Fanuc KAREL source: kb00041.KL

-- PROVISIONAL review KL for V1013-1; original PC SHA256 83256923c4522ad44c5b7a588ecc00707a52066454071d93bcafc420202dd29a
-- Incomplete behavior may be omitted. Consult companion uncertainty JSON. Do not deploy.
PROGRAM KB00041
%NOLOCKGROUP
BEGIN
  -- UNRESOLVED_PC offsets 5-14; opcodes 3F,75
  -- UNRESOLVED_PC offsets 19-30; opcodes 2E,23
  -- UNRESOLVED_PC offsets 35-53; opcodes 27,22,2A,22,31
  -- UNRESOLVED_PC offsets 58-62; opcodes 7F
END KB00041
